INTERFACE I_EventHandlers

END_INTERFACE

(* stored: Version 1.1.0.1, ProductVersion 3.1.4024.12
   Itf I_EventHandlers: Id {c2eecab6-598a-42dd-b6d3-99225444fbc7} *)
